TYPE "Handshake_ShW"
VERSION : 0.1
   STRUCT
      PLCOnline : Bool;
      PLCLive : Bool;
      ServerOnline : Int;
      ServerLiveBit : Int;
   END_STRUCT;

END_TYPE

